(* Logix 5000 project; controller L3 vendor 1 type 14 code 92 rev 20.12; software revision 20.04; part 6 of 9 *)
(* tags used below, declared in another part *)
   A_LVL_DEC : REAL;
   A_T_DEG : REAL;
   aux_cond_tour : REAL;
   AUX_LVL_DEC : REAL;
   B3 : DINT[100];
   cligno : BOOL;
   CONV_MSG_R_lancy : MESSAGE;
   CONV_MSG_W_lancy : MESSAGE;   // N9:70 dans n9:30
   F8 : REAL[100];
   FLOW_TOUR : DINT;
   I_R1 : REAL;
   I_R2 : REAL;
   I_R3 : REAL;
   I_R4 : REAL;
   INT_T_DEC : integrat;
   int_T_deg : integrat;
   L3_stat : DINT[20];
   LVL_ANO : REAL;
   LVL_COLMAT : REAL;
   N10 : DINT[233];
   N7 : DINT[200];
   N9 : DINT[200];   // niveau decapage vers lancy (n9[10) ;;N9[70]
   NCOM : INT[20];
   pmp_vid_colmat : BOOL;
   S_SP_T_COLMAT : DINT;
   s_T_2_DEC : REAL;
   S_T_DEC : DINT;
   scp_cond_tour : SCP;
   SCP_FLW_TOUR : SCP;
   scp_I_colo : SCP;
   scp_I_r1 : SCP;
   scp_I_r2 : SCP;
   scp_I_r3 : SCP;
   SCP_I_R4 : SCP;
   SCP_LVL_ANO : SCP;
   SCP_LVL_COLM : SCP;
   SCP_LVL_DEC : SCP;
   SCP_T_ANO : SCP;
   SCP_T_DEC : SCP;
   scp_T_deg : SCP;
   SCP_T_EAU_REFR : SCP;
   SCP_T_IN_COLM : SCP;
   SCP_T_MIL_COLM : SCP;
   SCP_T_OUT_COLM : SCP;
   SCP_TRACT : SCP;
   scp_u_colo : SCP;
   scp_u_r1 : SCP;
   scp_u_r2 : SCP;
   scp_u_r3 : SCP;
   SCP_U_R4 : SCP;
   stat_L3 : DINT[20];
   T4 : TIMER[180];
   T_EAU_REFROID : REAL;
   T_IN_COLMAT : DINT;
   T_MIL_COLMAT : REAL;
   t_minute : TIMER;   // tempo on toutes les minute
   T_OUT_COLMAT : REAL;
   test3 : REAL;
   test4 : DINT;
   test5 : DINT;
   TRACT : REAL;
   U_R1 : REAL;
   U_R2 : DINT;
   U_R3 : DINT;
   U_R4 : REAL;
(* _2_GENERAL, continued *)

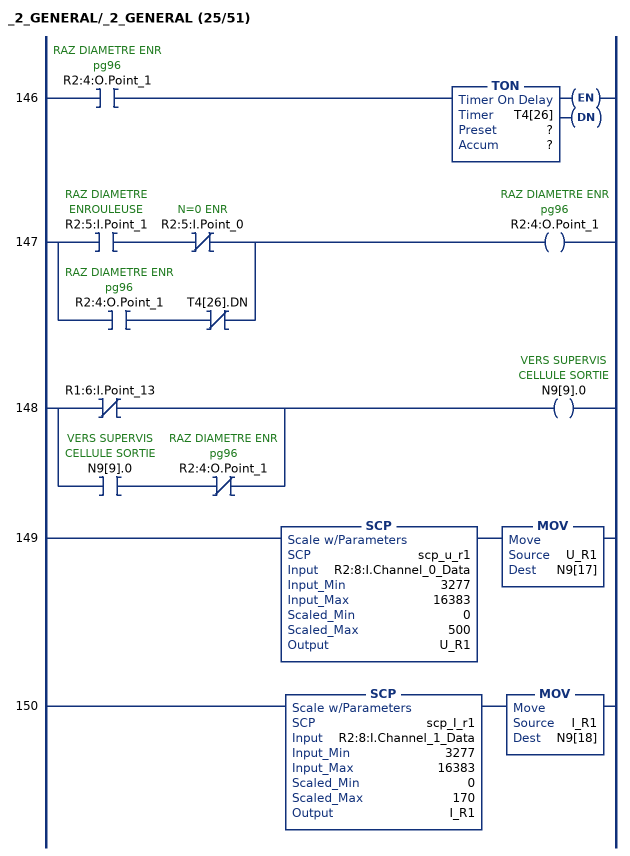
   146: XIC(R2:4:O.Point_1)TON(T4[26],?,?);
   147: [XIC(R2:5:I.Point_1) XIO(R2:5:I.Point_0) ,XIC(R2:4:O.Point_1) XIO(T4[26].DN) ]OTE(R2:4:O.Point_1);
   148: [XIO(R1:6:I.Point_13) ,XIC(N9[9].0) XIO(R2:4:O.Point_1) ]OTE(N9[9].0);
   149: SCP(scp_u_r1,R2:8:I.Channel_0_Data,3277,16383,0,500,U_R1)MOV(U_R1,N9[17]);
   150: SCP(scp_I_r1,R2:8:I.Channel_1_Data,3277,16383,0,170,I_R1)MOV(I_R1,N9[18]);
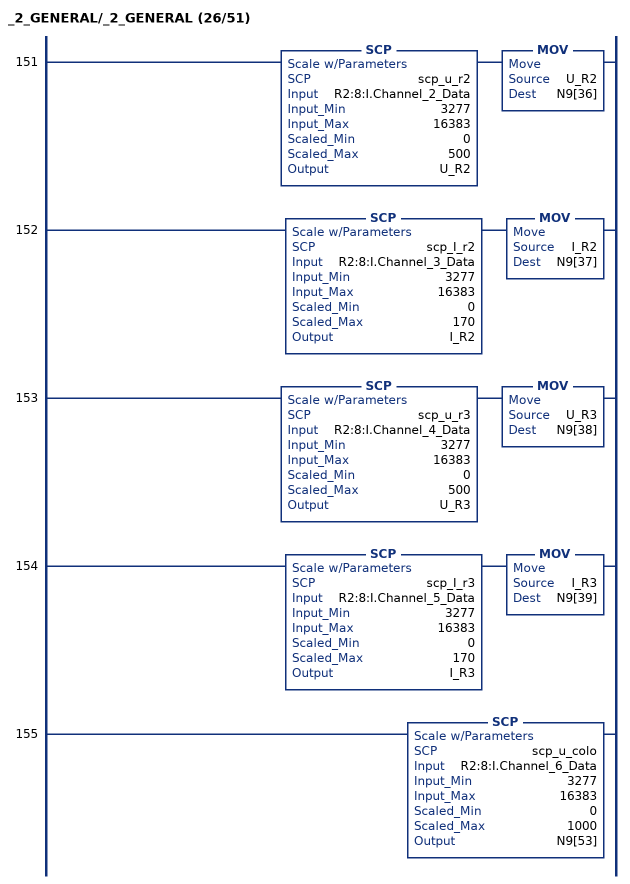
   151: SCP(scp_u_r2,R2:8:I.Channel_2_Data,3277,16383,0,500,U_R2)MOV(U_R2,N9[36]);
   152: SCP(scp_I_r2,R2:8:I.Channel_3_Data,3277,16383,0,170,I_R2)MOV(I_R2,N9[37]);
   153: SCP(scp_u_r3,R2:8:I.Channel_4_Data,3277,16383,0,500,U_R3)MOV(U_R3,N9[38]);
   154: SCP(scp_I_r3,R2:8:I.Channel_5_Data,3277,16383,0,170,I_R3)MOV(I_R3,N9[39]);
   155: SCP(scp_u_colo,R2:8:I.Channel_6_Data,3277,16383,0,1000,N9[53]);
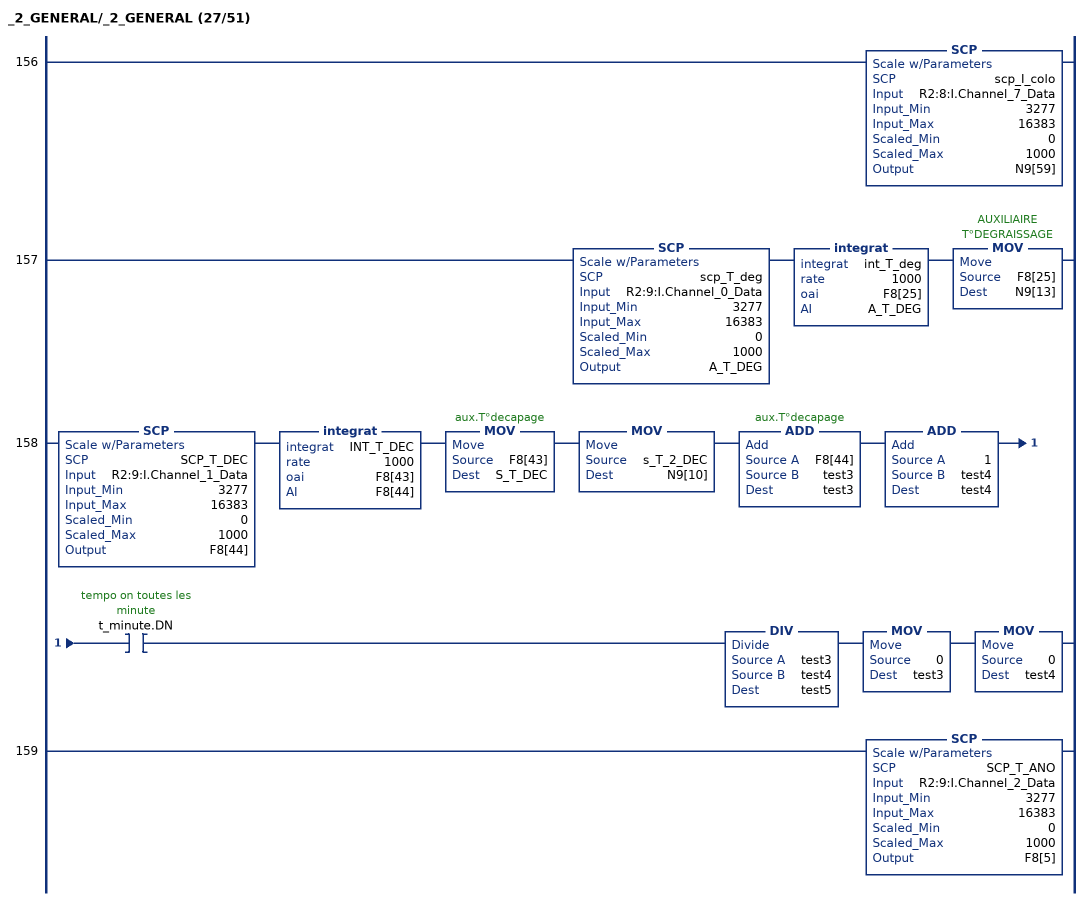
   156: SCP(scp_I_colo,R2:8:I.Channel_7_Data,3277,16383,0,1000,N9[59]);
   157: SCP(scp_T_deg,R2:9:I.Channel_0_Data,3277,16383,0,1000,A_T_DEG)integrat(int_T_deg,1000,F8[25],A_T_DEG)MOV(F8[25],N9[13]);
   158: SCP(SCP_T_DEC,R2:9:I.Channel_1_Data,3277,16383,0,1000,F8[44])integrat(INT_T_DEC,1000,F8[43],F8[44])MOV(F8[43],S_T_DEC)MOV(s_T_2_DEC,N9[10])ADD(F8[44],test3,test3)ADD(1,test4,test4)XIC(t_minute.DN)DIV(test3,test4,test5)MOV(0,test3)MOV(0,test4);
   159: SCP(SCP_T_ANO,R2:9:I.Channel_2_Data,3277,16383,0,1000,F8[5]);
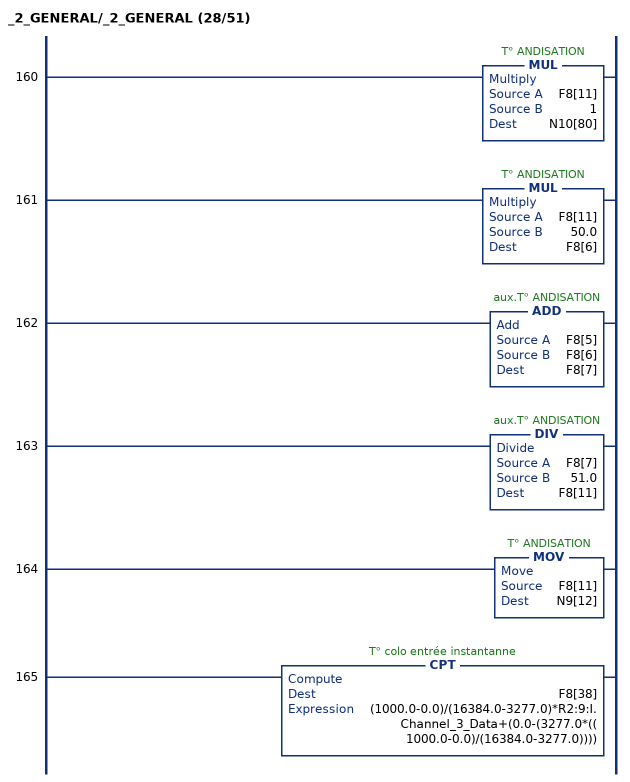
   160: MUL(F8[11],1,N10[80]);
   161: MUL(F8[11],50.0,F8[6]);
   162: ADD(F8[5],F8[6],F8[7]);
   163: DIV(F8[7],51.0,F8[11]);
   164: MOV(F8[11],N9[12]);
   165: CPT(F8[38],(1000.0-0.0)/(16384.0-3277.0)*R2:9:I.Channel_3_Data+(0.0-(3277.0*((1000.0-0.0)/(16384.0-3277.0)))));
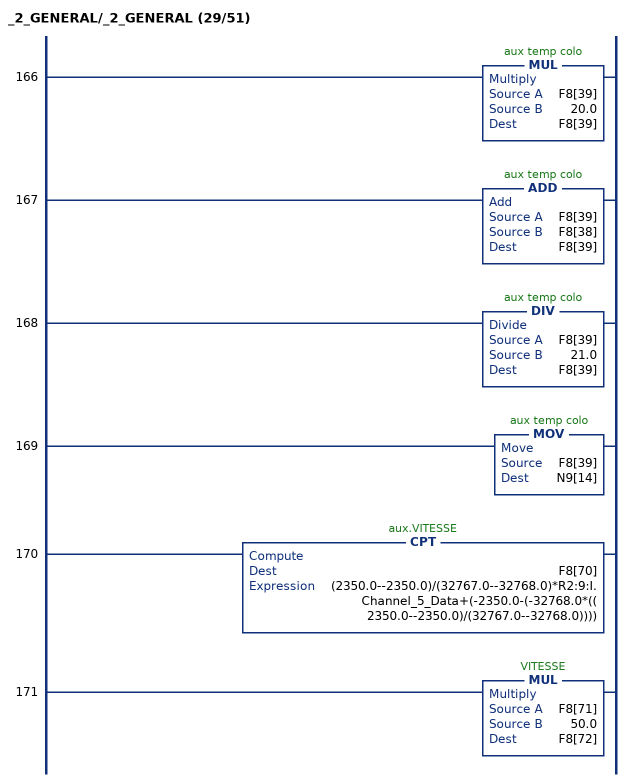
   166: MUL(F8[39],20.0,F8[39]);
   167: ADD(F8[39],F8[38],F8[39]);
   168: DIV(F8[39],21.0,F8[39]);
   169: MOV(F8[39],N9[14]);
   170: CPT(F8[70],(2350.0--2350.0)/(32767.0--32768.0)*R2:9:I.Channel_5_Data+(-2350.0-(-32768.0*((2350.0--2350.0)/(32767.0--32768.0)))));
   171: MUL(F8[71],50.0,F8[72]);
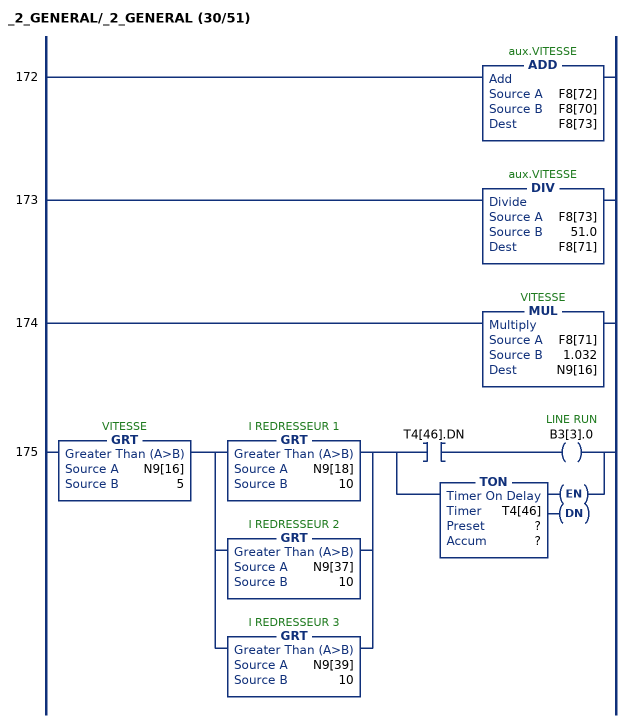
   172: ADD(F8[72],F8[70],F8[73]);
   173: DIV(F8[73],51.0,F8[71]);
   174: MUL(F8[71],1.032,N9[16]);
   175: GRT(N9[16],5)[GRT(N9[18],10) ,GRT(N9[37],10) ,GRT(N9[39],10) ][XIC(T4[46].DN) OTE(B3[3].0) ,TON(T4[46],?,?) ];
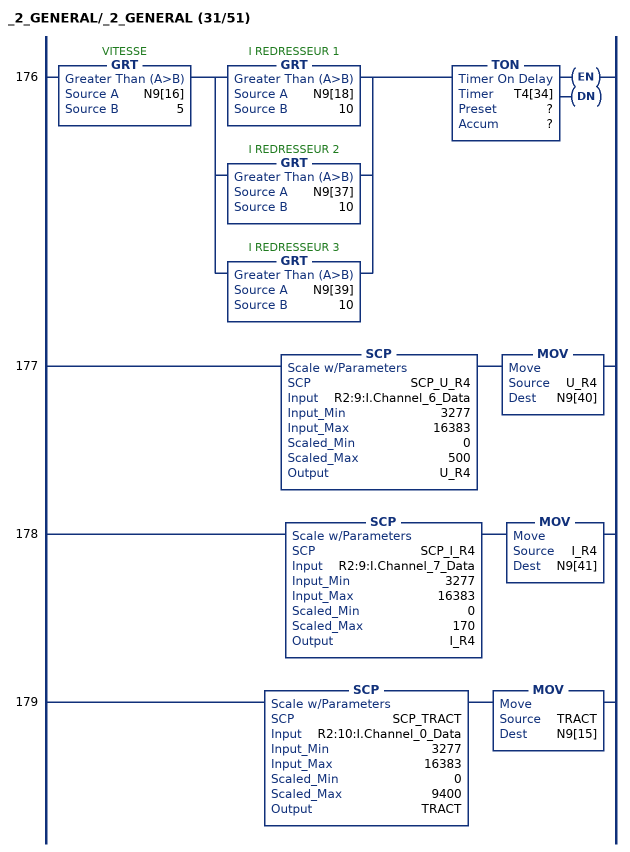
   176: GRT(N9[16],5)[GRT(N9[18],10) ,GRT(N9[37],10) ,GRT(N9[39],10) ]TON(T4[34],?,?);
   177: SCP(SCP_U_R4,R2:9:I.Channel_6_Data,3277,16383,0,500,U_R4)MOV(U_R4,N9[40]);
   178: SCP(SCP_I_R4,R2:9:I.Channel_7_Data,3277,16383,0,170,I_R4)MOV(I_R4,N9[41]);
   179: SCP(SCP_TRACT,R2:10:I.Channel_0_Data,3277,16383,0,9400,TRACT)MOV(TRACT,N9[15]);
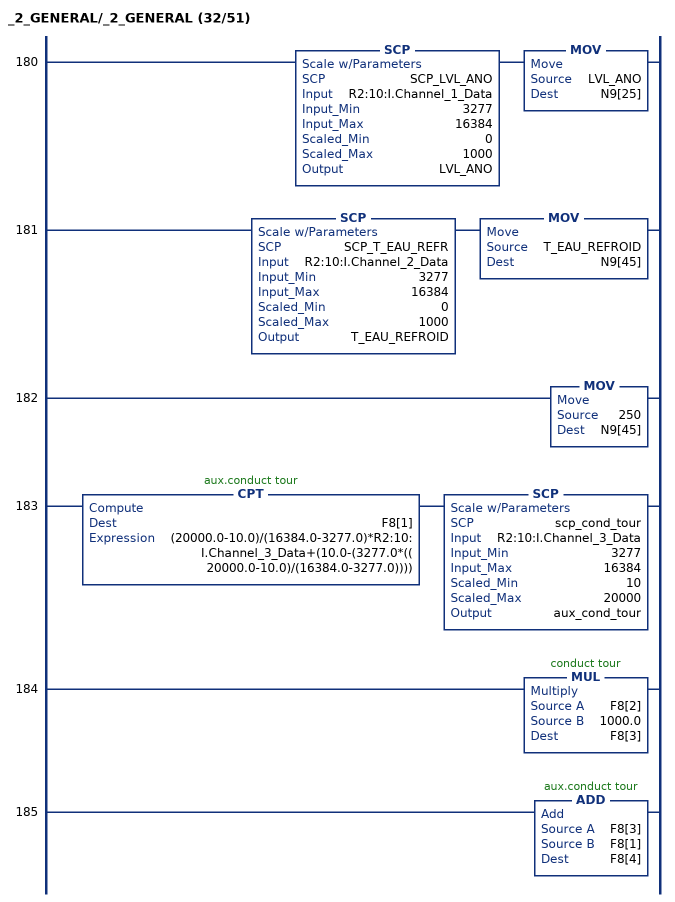
   180: SCP(SCP_LVL_ANO,R2:10:I.Channel_1_Data,3277,16384,0,1000,LVL_ANO)MOV(LVL_ANO,N9[25]);
   181: SCP(SCP_T_EAU_REFR,R2:10:I.Channel_2_Data,3277,16384,0,1000,T_EAU_REFROID)MOV(T_EAU_REFROID,N9[45]);
   182: MOV(250,N9[45]);
   183: CPT(F8[1],(20000.0-10.0)/(16384.0-3277.0)*R2:10:I.Channel_3_Data+(10.0-(3277.0*((20000.0-10.0)/(16384.0-3277.0)))))SCP(scp_cond_tour,R2:10:I.Channel_3_Data,3277,16384,10,20000,aux_cond_tour);
   184: MUL(F8[2],1000.0,F8[3]);
   185: ADD(F8[3],F8[1],F8[4]);
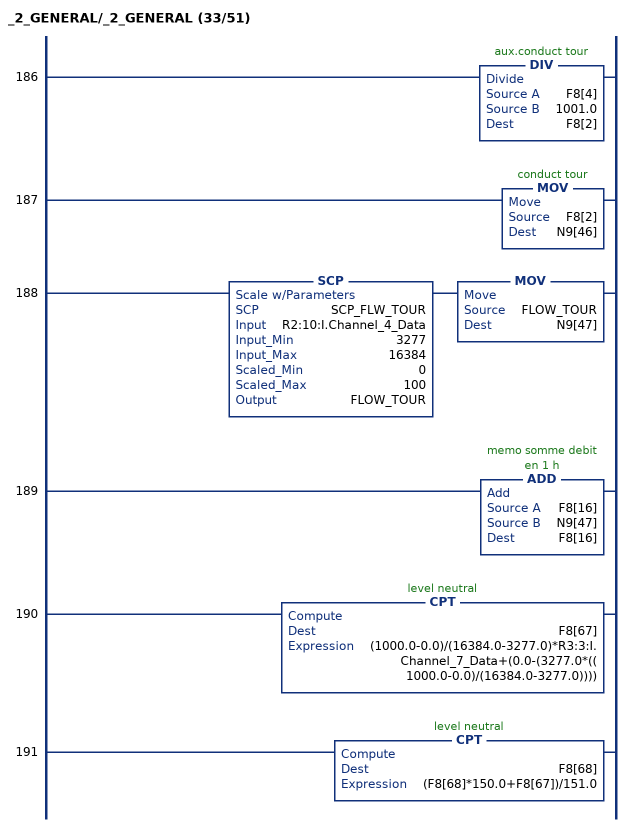
   186: DIV(F8[4],1001.0,F8[2]);
   187: MOV(F8[2],N9[46]);
   188: SCP(SCP_FLW_TOUR,R2:10:I.Channel_4_Data,3277,16384,0,100,FLOW_TOUR)MOV(FLOW_TOUR,N9[47]);
   189: ADD(F8[16],N9[47],F8[16]);
   190: CPT(F8[67],(1000.0-0.0)/(16384.0-3277.0)*R3:3:I.Channel_7_Data+(0.0-(3277.0*((1000.0-0.0)/(16384.0-3277.0)))));
   191: CPT(F8[68],(F8[68]*150.0+F8[67])/151.0);
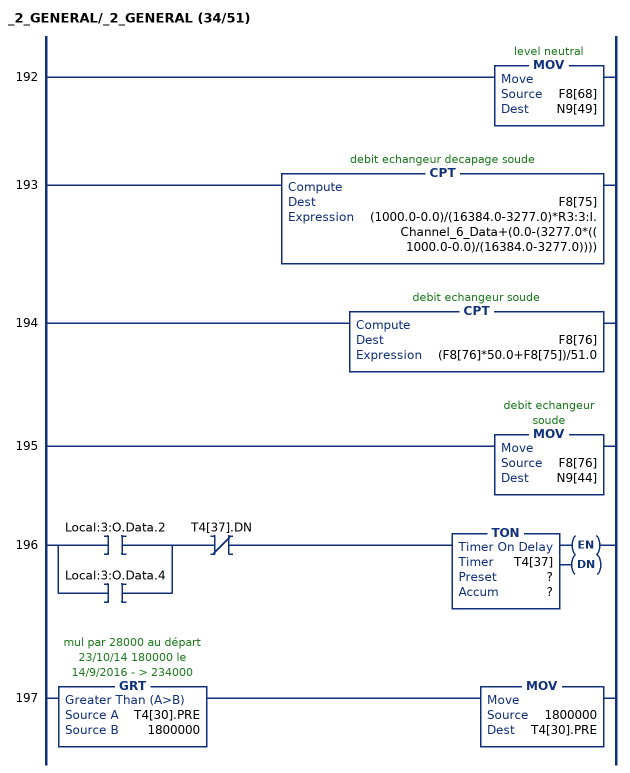
   192: MOV(F8[68],N9[49]);
   193: CPT(F8[75],(1000.0-0.0)/(16384.0-3277.0)*R3:3:I.Channel_6_Data+(0.0-(3277.0*((1000.0-0.0)/(16384.0-3277.0)))));
   194: CPT(F8[76],(F8[76]*50.0+F8[75])/51.0);
   195: MOV(F8[76],N9[44]);
   196: [XIC(Local:3:O.Data.2) ,XIC(Local:3:O.Data.4) ]XIO(T4[37].DN)TON(T4[37],?,?);
   197: GRT(T4[30].PRE,1800000)MOV(1800000,T4[30].PRE);
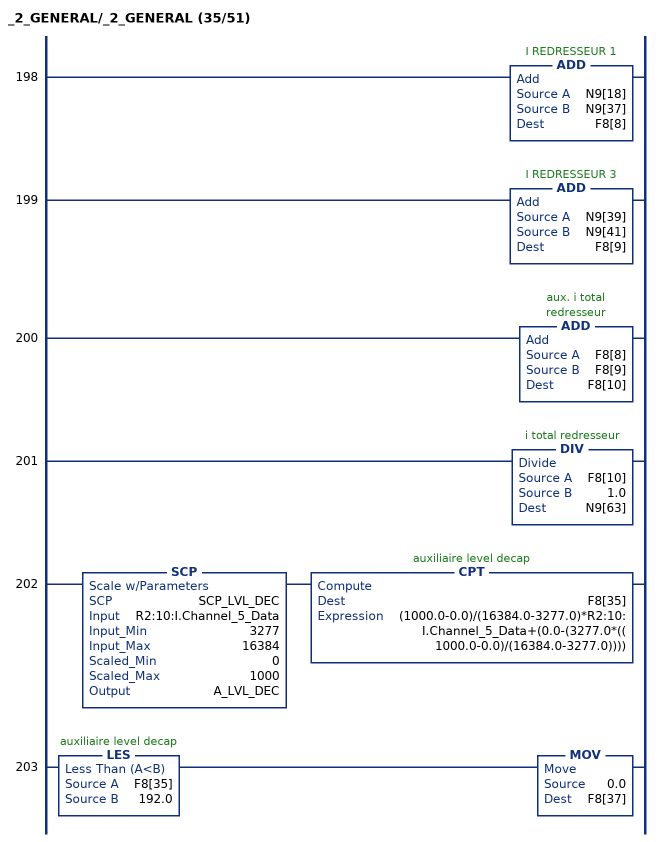
   198: ADD(N9[18],N9[37],F8[8]);
   199: ADD(N9[39],N9[41],F8[9]);
   200: ADD(F8[8],F8[9],F8[10]);
   201: DIV(F8[10],1.0,N9[63]);
   202: SCP(SCP_LVL_DEC,R2:10:I.Channel_5_Data,3277,16384,0,1000,A_LVL_DEC)CPT(F8[35],(1000.0-0.0)/(16384.0-3277.0)*R2:10:I.Channel_5_Data+(0.0-(3277.0*((1000.0-0.0)/(16384.0-3277.0)))));
   203: LES(F8[35],192.0)MOV(0.0,F8[37]);
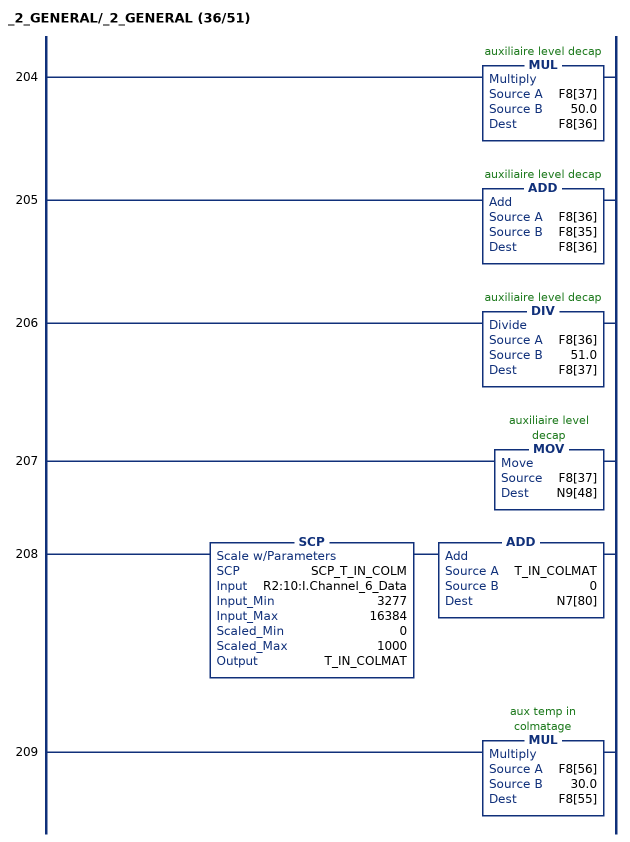
   204: MUL(F8[37],50.0,F8[36]);
   205: ADD(F8[36],F8[35],F8[36]);
   206: DIV(F8[36],51.0,F8[37]);
   207: MOV(F8[37],N9[48]);
   208: SCP(SCP_T_IN_COLM,R2:10:I.Channel_6_Data,3277,16384,0,1000,T_IN_COLMAT)ADD(T_IN_COLMAT,0,N7[80]);
   209: MUL(F8[56],30.0,F8[55]);
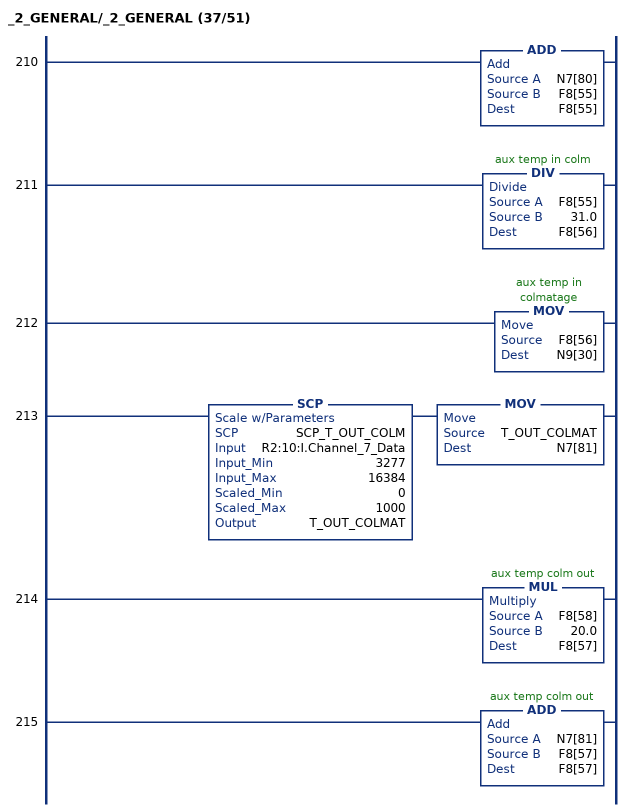
   210: ADD(N7[80],F8[55],F8[55]);
   211: DIV(F8[55],31.0,F8[56]);
   212: MOV(F8[56],N9[30]);
   213: SCP(SCP_T_OUT_COLM,R2:10:I.Channel_7_Data,3277,16384,0,1000,T_OUT_COLMAT)MOV(T_OUT_COLMAT,N7[81]);
   214: MUL(F8[58],20.0,F8[57]);
   215: ADD(N7[81],F8[57],F8[57]);
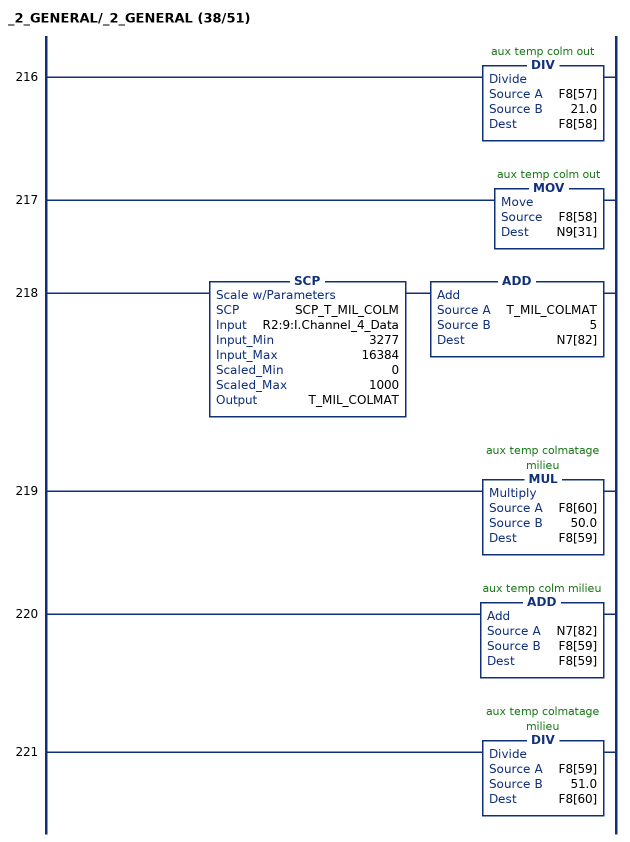
   216: DIV(F8[57],21.0,F8[58]);
   217: MOV(F8[58],N9[31]);
   218: SCP(SCP_T_MIL_COLM,R2:9:I.Channel_4_Data,3277,16384,0,1000,T_MIL_COLMAT)ADD(T_MIL_COLMAT,5,N7[82]);
   219: MUL(F8[60],50.0,F8[59]);
   220: ADD(N7[82],F8[59],F8[59]);
   221: DIV(F8[59],51.0,F8[60]);
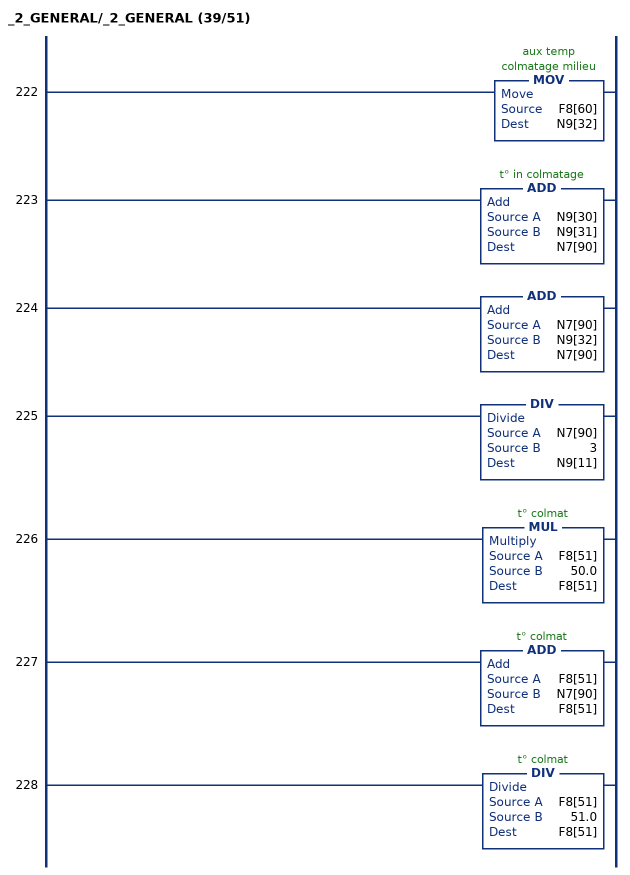
   222: MOV(F8[60],N9[32]);
   223: ADD(N9[30],N9[31],N7[90]);
   224: ADD(N7[90],N9[32],N7[90]);
   225: DIV(N7[90],3,N9[11]);
   226: MUL(F8[51],50.0,F8[51]);
   227: ADD(F8[51],N7[90],F8[51]);
   228: DIV(F8[51],51.0,F8[51]);
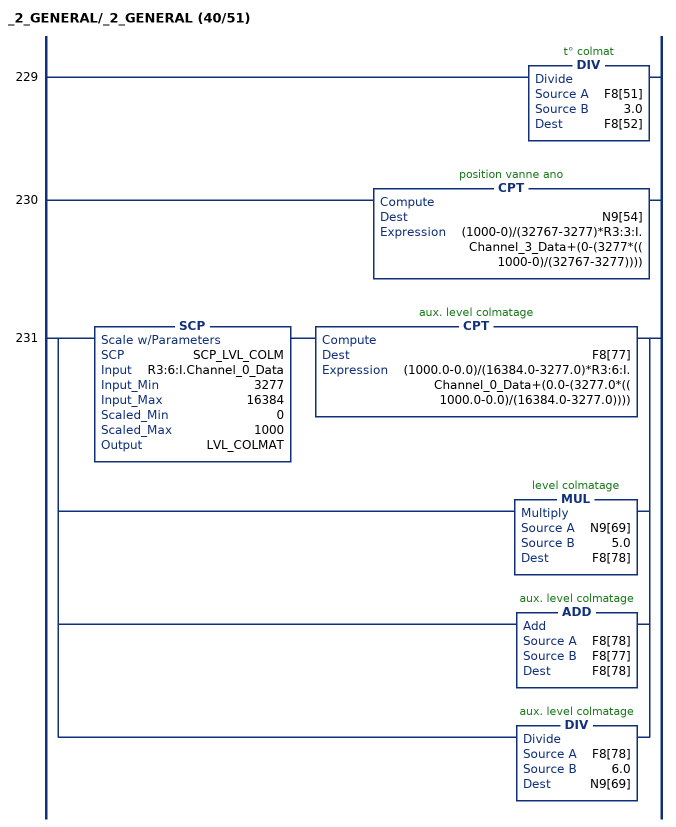
   229: DIV(F8[51],3.0,F8[52]);
   230: CPT(N9[54],(1000-0)/(32767-3277)*R3:3:I.Channel_3_Data+(0-(3277*((1000-0)/(32767-3277)))));
   231: [SCP(SCP_LVL_COLM,R3:6:I.Channel_0_Data,3277,16384,0,1000,LVL_COLMAT) CPT(F8[77],(1000.0-0.0)/(16384.0-3277.0)*R3:6:I.Channel_0_Data+(0.0-(3277.0*((1000.0-0.0)/(16384.0-3277.0))))) ,MUL(N9[69],5.0,F8[78]) ,ADD(F8[78],F8[77],F8[78]) ,DIV(F8[78],6.0,N9[69]) ];
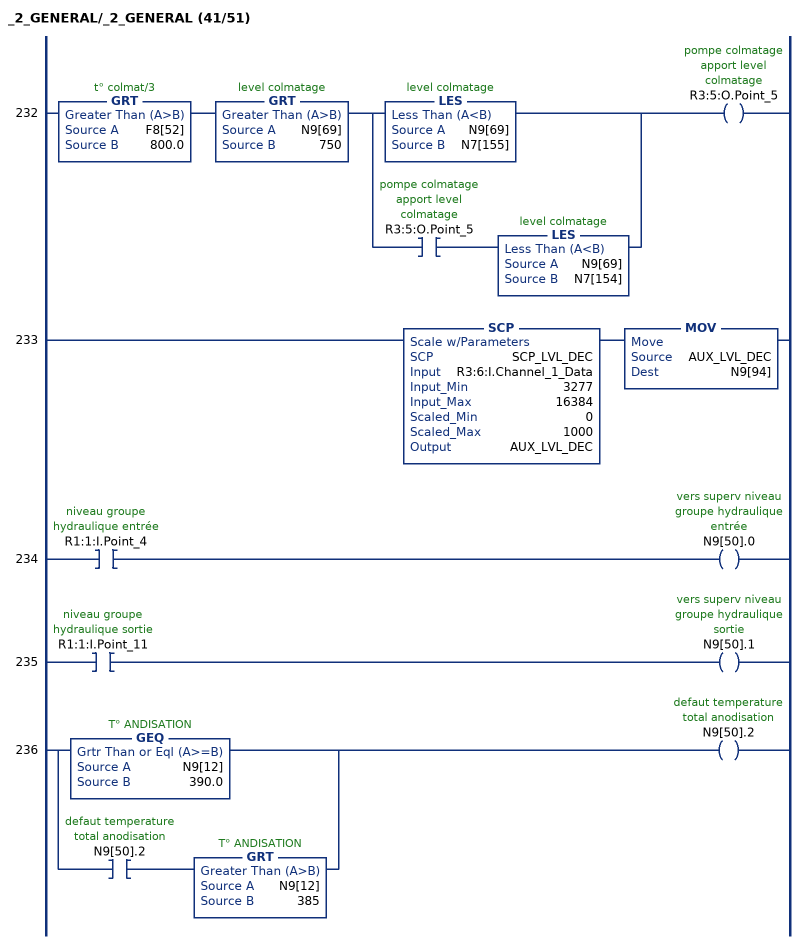
   232: GRT(F8[52],800.0)GRT(N9[69],750)[LES(N9[69],N7[155]) ,XIC(R3:5:O.Point_5) LES(N9[69],N7[154]) ]OTE(R3:5:O.Point_5);
   233: SCP(SCP_LVL_DEC,R3:6:I.Channel_1_Data,3277,16384,0,1000,AUX_LVL_DEC)MOV(AUX_LVL_DEC,N9[94]);
   234: XIC(R1:1:I.Point_4)OTE(N9[50].0);
   235: XIC(R1:1:I.Point_11)OTE(N9[50].1);
   236: [GEQ(N9[12],390.0) ,XIC(N9[50].2) GRT(N9[12],385) ]OTE(N9[50].2);
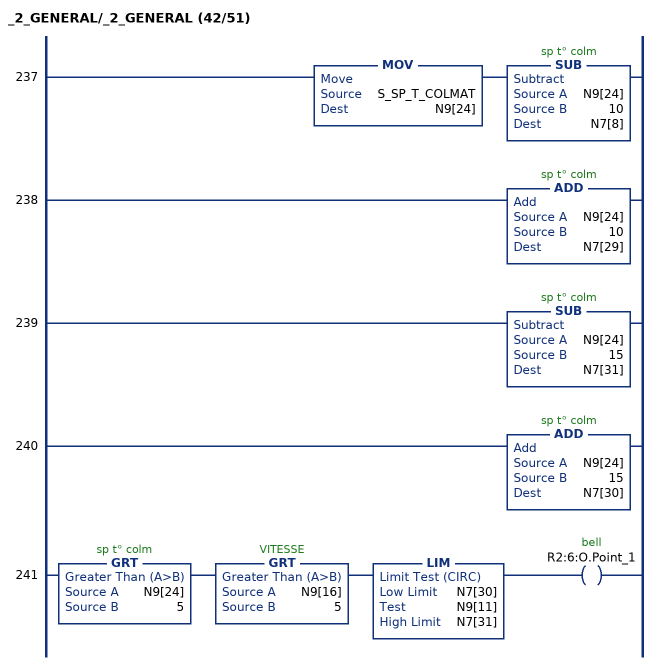
   237: MOV(S_SP_T_COLMAT,N9[24])SUB(N9[24],10,N7[8]);
   238: ADD(N9[24],10,N7[29]);
   239: SUB(N9[24],15,N7[31]);
   240: ADD(N9[24],15,N7[30]);
   241: GRT(N9[24],5)GRT(N9[16],5)LIM(N7[30],N9[11],N7[31])OTE(R2:6:O.Point_1);
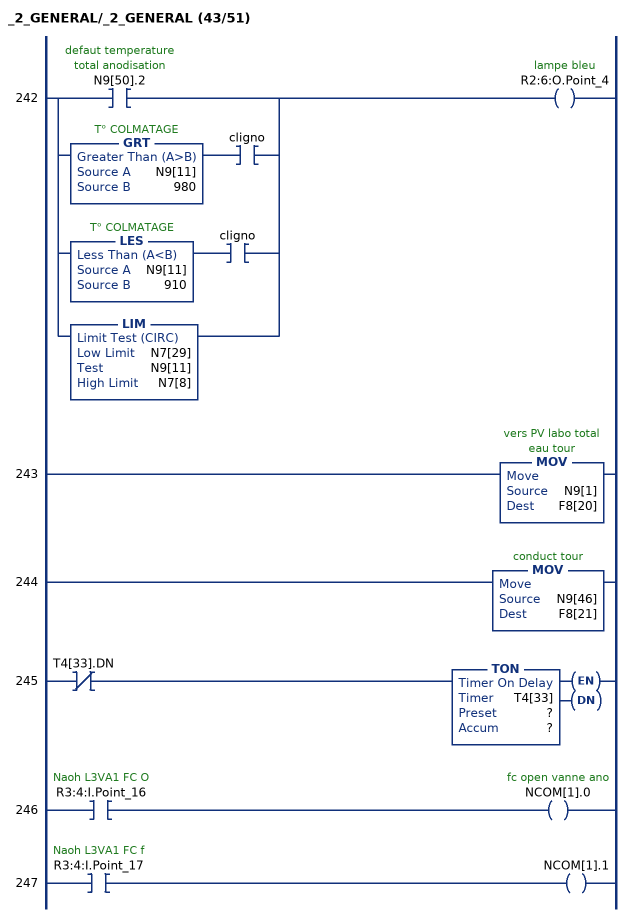
   242: [XIC(N9[50].2) ,GRT(N9[11],980) XIC(cligno) ,LES(N9[11],910) XIC(cligno) ,LIM(N7[29],N9[11],N7[8]) ]OTE(R2:6:O.Point_4);
   243: MOV(N9[1],F8[20]);
   244: MOV(N9[46],F8[21]);
   245: XIO(T4[33].DN)TON(T4[33],?,?);
   246: XIC(R3:4:I.Point_16)OTE(NCOM[1].0);
   247: XIC(R3:4:I.Point_17)OTE(NCOM[1].1);
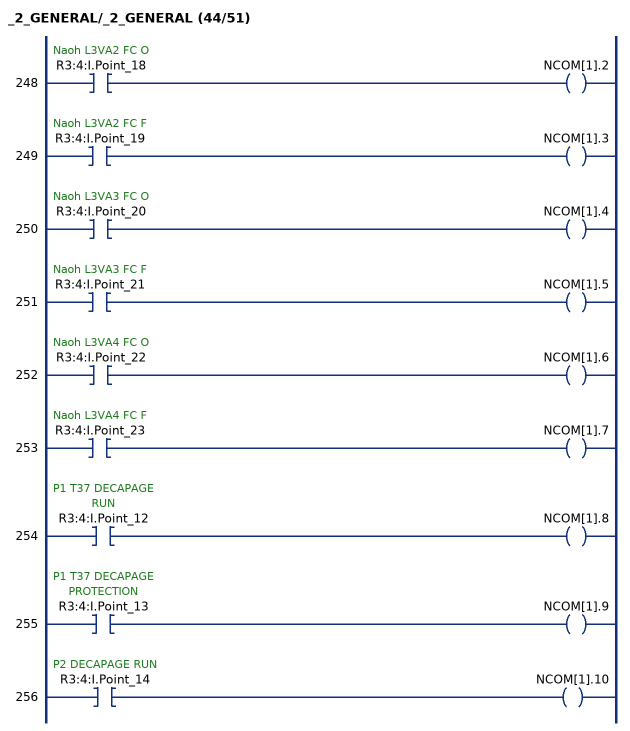
   248: XIC(R3:4:I.Point_18)OTE(NCOM[1].2);
   249: XIC(R3:4:I.Point_19)OTE(NCOM[1].3);
   250: XIC(R3:4:I.Point_20)OTE(NCOM[1].4);
   251: XIC(R3:4:I.Point_21)OTE(NCOM[1].5);
   252: XIC(R3:4:I.Point_22)OTE(NCOM[1].6);
   253: XIC(R3:4:I.Point_23)OTE(NCOM[1].7);
   254: XIC(R3:4:I.Point_12)OTE(NCOM[1].8);
   255: XIC(R3:4:I.Point_13)OTE(NCOM[1].9);
   256: XIC(R3:4:I.Point_14)OTE(NCOM[1].10);
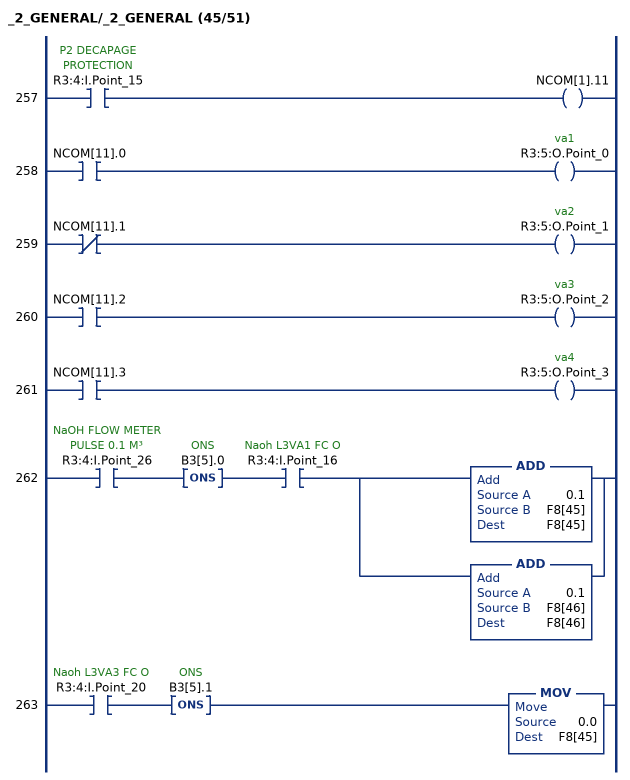
   257: XIC(R3:4:I.Point_15)OTE(NCOM[1].11);
   258: XIC(NCOM[11].0)OTE(R3:5:O.Point_0);
   259: XIO(NCOM[11].1)OTE(R3:5:O.Point_1);
   260: XIC(NCOM[11].2)OTE(R3:5:O.Point_2);
   261: XIC(NCOM[11].3)OTE(R3:5:O.Point_3);
   262: XIC(R3:4:I.Point_26)ONS(B3[5].0)XIC(R3:4:I.Point_16)[ADD(0.1,F8[45],F8[45]) ,ADD(0.1,F8[46],F8[46]) ];
   263: XIC(R3:4:I.Point_20)ONS(B3[5].1)MOV(0.0,F8[45]);
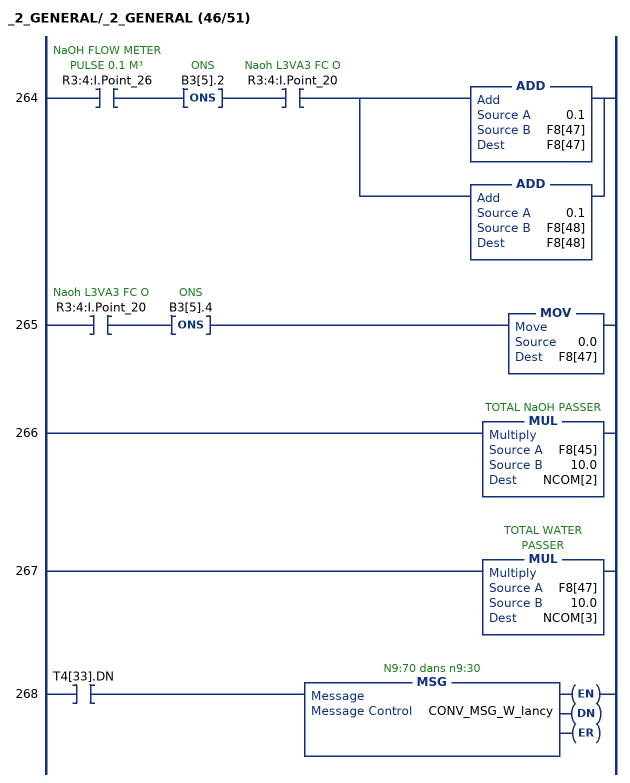
   264: XIC(R3:4:I.Point_26)ONS(B3[5].2)XIC(R3:4:I.Point_20)[ADD(0.1,F8[47],F8[47]) ,ADD(0.1,F8[48],F8[48]) ];
   265: XIC(R3:4:I.Point_20)ONS(B3[5].4)MOV(0.0,F8[47]);
   266: MUL(F8[45],10.0,NCOM[2]);
   267: MUL(F8[47],10.0,NCOM[3]);
   268: XIC(T4[33].DN)MSG(CONV_MSG_W_lancy);
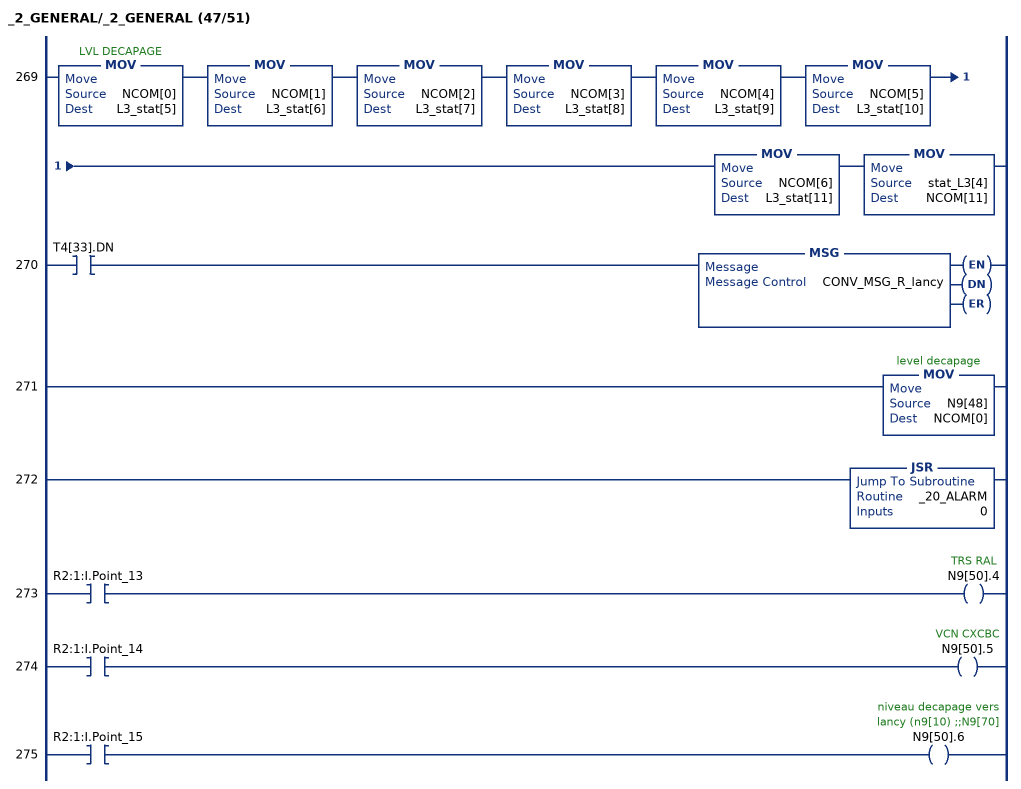
   269: MOV(NCOM[0],L3_stat[5])MOV(NCOM[1],L3_stat[6])MOV(NCOM[2],L3_stat[7])MOV(NCOM[3],L3_stat[8])MOV(NCOM[4],L3_stat[9])MOV(NCOM[5],L3_stat[10])MOV(NCOM[6],L3_stat[11])MOV(stat_L3[4],NCOM[11]);
   270: XIC(T4[33].DN)MSG(CONV_MSG_R_lancy);
   271: MOV(N9[48],NCOM[0]);
   272: JSR(_20_ALARM,0);
   273: XIC(R2:1:I.Point_13)OTE(N9[50].4);
   274: XIC(R2:1:I.Point_14)OTE(N9[50].5);
   275: XIC(R2:1:I.Point_15)OTE(N9[50].6);
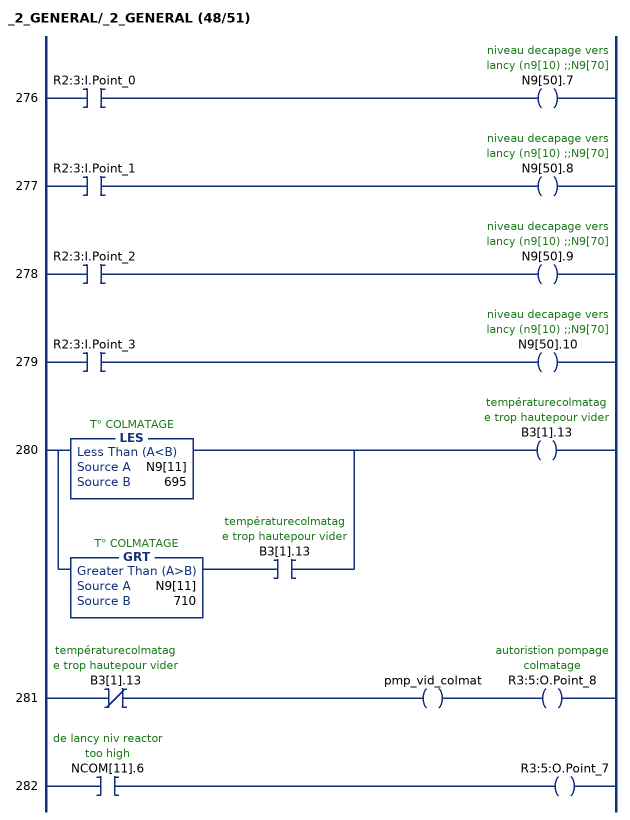
   276: XIC(R2:3:I.Point_0)OTE(N9[50].7);
   277: XIC(R2:3:I.Point_1)OTE(N9[50].8);
   278: XIC(R2:3:I.Point_2)OTE(N9[50].9);
   279: XIC(R2:3:I.Point_3)OTE(N9[50].10);
   280: [LES(N9[11],695) ,GRT(N9[11],710) XIC(B3[1].13) ]OTE(B3[1].13);
   281: XIO(B3[1].13)OTE(pmp_vid_colmat)OTE(R3:5:O.Point_8);
   282: XIC(NCOM[11].6)OTE(R3:5:O.Point_7);
